ABB RAPID module: Wobj_work2E2e.MOD

MODULE Wobj_work2E2e
	! Points are read in order of declaration.
  ! Please do not change the order of points!

  LOCAL PERS robtarget pWobj_O_PointX1:=[[-652.9529,-386.9818,314.64],[0.147992044687271,0.850937187671661,0.318506091833115,-0.390587002038956],[-2,0,-1,0],[9E+09,9E+09,9E+09,9E+09,9E+09,9E+09]];
	LOCAL PERS robtarget pWobj_O_PointX2:=[[-504.5624,-393.7464,306.0317],[0.147958293557167,0.850943028926849,0.31852525472641,-0.390571355819702],[-2,0,-1,0],[9E+09,9E+09,9E+09,9E+09,9E+09,9E+09]];
	LOCAL PERS robtarget pWobj_O_PointY1:=[[-658.44,-196.9807,312.2636],[0.147940367460251,0.851009845733643,0.318539261817932,-0.390421092510223],[-2,0,-1,0],[9E+09,9E+09,9E+09,9E+09,9E+09,9E+09]];

ENDMODULE
